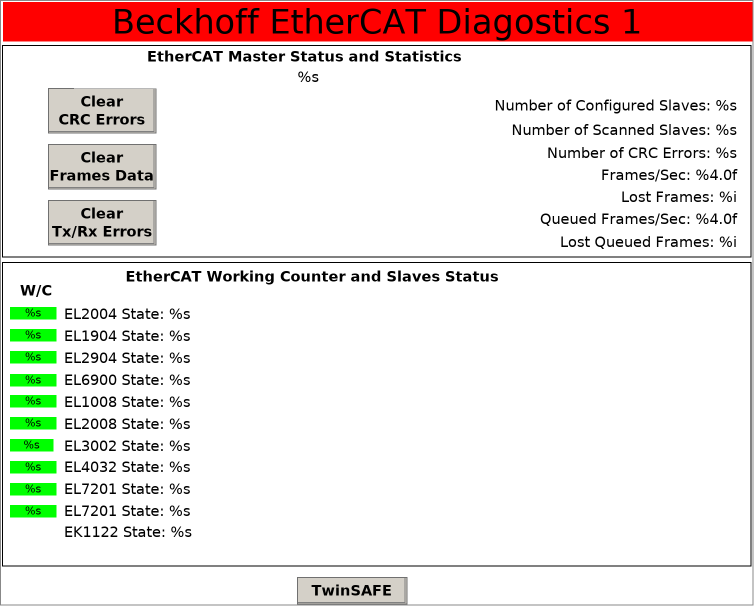
VISUALIZATION EtherCAT_Diag1  // 754x606
    Button (297,577 110x27), "TwinSAFE"
        OnMouseClick: change screen: TwinSAFE
    RoundedRectangle (3,2 749x39), "Beckhoff EtherCAT Diagostics 1"
    RoundedRectangle (2,45 749x212)
    RoundedRectangle (2,262 749x304)
    Label (152,45 305x23), "EtherCAT Master Status and Statistics"
    Button (48,88 108x45), "Clear CRC Errors"
        tap g_xHMI_CearMFStatCRCs
    Label (123,265 378x23), "EtherCAT Working Counter and Slaves Status"
    Button (48,144 108x45), "Clear Frames Data"
        tap g_xHMI_ClearMFStatFrames
    Button (48,200 108x45), "Clear Tx/Rx Errors"
        tap g_xHMI_ClearMFStatTxRxErr
    Label (14,279 44x23), "W/C"
    Rectangle (74,66 469x22), "%s", text variable: g_sHMI_StateMaster
    Rectangle (428,97 312x17), "Number of Configured Slaves: %s", text variable: g_uiHMI_ConfSlaves
    Rectangle (429,121 311x18), "Number of Scanned Slaves: %s", text variable: g_uiHMI_ScannedSlaves
    Rectangle (430,144 310x18), "Number of CRC Errors: %s", text variable: g_dwHMI_TotalCrcErrors
    Rectangle (431,166 309x18), "Frames/Sec: %4.0f", text variable: g_lrHMI_FramesPerSecond
    Rectangle (430,188 310x18), "Lost Frames: %i", text variable: g_udiHMI_LostFrames
    Rectangle (431,210 309x18), "Queued Frames/Sec: %4.0f", text variable: g_lrHMI_QueuedFramesPerSecond
    Rectangle (432,233 308x18), "Lost Queued Frames: %i", text variable: g_udiHMI_LostQueuedFrames
    Rectangle (61,303 686x22), "EL2004 State: %s", text variable: g_sHMI_StateEL2004
    Rectangle (61,325 685x22), "EL1904 State: %s", text variable: g_sHMI_StateEL1904
    Rectangle (61,347 686x22), "EL2904 State: %s", text variable: g_sHMI_StateEL2904
    Rectangle (61,369 684x22), "EL6900 State: %s", text variable: g_sHMI_StateEL6900
    Rectangle (61,391 683x22), "EL1008 State: %s", text variable: g_sHMI_StateEL1008
    Rectangle (61,413 685x22), "EL2008 State: %s", text variable: g_sHMI_StateEL2008
    Rectangle (61,435 685x22), "EL3002 State: %s", text variable: g_sHMI_StateEL3002
    Rectangle (61,456 684x22), "EL4032 State: %s", text variable: g_sHMI_StateEL4032
    Rectangle (10,307 46x12), "%s", text variable: g_xEL2004_Wc
    Rectangle (10,329 46x12), "%s", text variable: g_xEL1904_Wc
    Rectangle (10,351 46x12), "%s", text variable: g_xEL2904_Wc
    Rectangle (10,374 46x12), "%s", text variable: g_xEL6900_Wc
    Rectangle (10,395 46x12), "%s", text variable: g_xEL1008_Wc
    Rectangle (10,417 46x12), "%s", text variable: g_xEL2008_Wc
    Rectangle (10,439 43x12), "%s", text variable: g_xEL3002_Wc
    Rectangle (10,461 46x12), "%s", text variable: g_xEL4032_Wc
    Rectangle (61,478 684x22), "EL7201 State: %s", text variable: g_sHMI_StateEL7201_1
    Rectangle (10,483 46x12), "%s", text variable: g_xEL7201_2_Wc
    Rectangle (61,500 684x22), "EL7201 State: %s", text variable: g_sHMI_StateEL7201_2
    Rectangle (10,505 46x12), "%s", text variable: g_xEL7201_2_Wc
    Rectangle (61,521 684x22), "EK1122 State: %s", text variable: g_sHMI_StateEK1122
END_VISUALIZATION

(* stored: Version 1.1.0.1, ProductVersion 3.1.0.18
   Visu EtherCAT_Diag1: Id {e106253d-815d-4bb5-9cde-fb194eb0b815} *)
